(* Logix 5000 project; controller VET 1756-L62 rev 19.52; software revision 19.01; part 22 of 27 *)
(* tags used below, declared in another part *)
   _reset_local : ALIAS FOR _reset_locales.0;
   batch_in : batch;
   batch_out : batch;
   db1_var_batch : variables_procedimientos;
   db3_var_rep : variables_procedimientos;
   var_wd : variables_procedimientos;
   _Eqp_Cfg : Eqp_Cfg[800];
   Batch : batch[10];
   borrar : DINT[100];
   DRT : DRTs[10];
   simulacion : BOOL;
   TabBin : Bins_Setup;
   Timer : TIMER[500];
   vdf : VDFS[20];
(* Main, continued *)

ROUTINE main   (* ladder *)
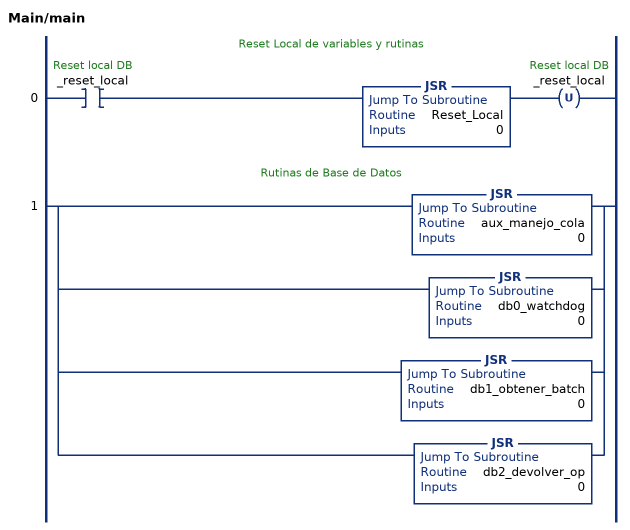
   // Reset Local de variables y rutinas
   0: XIC(_reset_local)JSR(Reset_Local,0)OTU(_reset_local);
   // Rutinas de Base de Datos
   1: [JSR(aux_manejo_cola,0) ,JSR(db0_watchdog,0) ,JSR(db1_obtener_batch,0) ,JSR(db2_devolver_op,0) ];
END_ROUTINE

ROUTINE Reset_Local   (* ladder *)
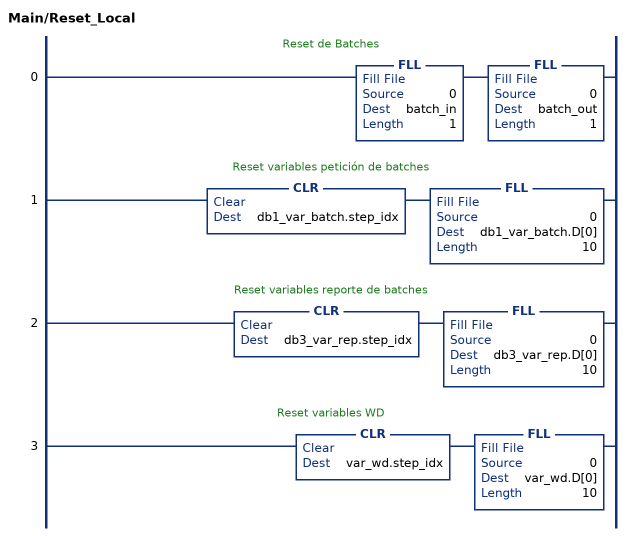
   // Reset de Batches
   0: FLL(0,batch_in,1)FLL(0,batch_out,1);
   // Reset variables petición de batches
   1: CLR(db1_var_batch.step_idx)FLL(0,db1_var_batch.D[0],10);
   // Reset variables reporte de batches
   2: CLR(db3_var_rep.step_idx)FLL(0,db3_var_rep.D[0],10);
   // Reset variables WD
   3: CLR(var_wd.step_idx)FLL(0,var_wd.D[0],10);
END_ROUTINE
END_PROGRAM

PROGRAM Main1   (* main routine Main, fault routine Error_Handler *)
VAR
   Automatismos : DINT := 7;
   Aux : DINT[500] := ([0] := 2014, [1] := 5, [2] := 15, [3] := 18, [4] := 46, [5] := 49, [6] := 20121005, [7] := 1184649, [8] := 1335329064, [9] := 2097152, [10] := 310798972, [11] := 326008, [13] := 1073741824, [14] := 4, [15] := 100, [16] := 180, [17] := 180, [18] := -25306, [19] := 1000000000, [20] := 1000000000, [21] := 1000000, [22] := 1099, [25] := 3, [27] := 164, [28] := 6347, [30] := 32, [34] := 111, [35] := 27, [36] := 10, [38] := 9, [45] := 4, [46] := 420, [47] := 14, [49] := 15999, [51] := 1, [52] := 10, [53] := 1, [54] := 1, [55] := 2, [56] := 47, [57] := 5, [58] := 6, [61] := 10, [62] := 1, [63] := 60, [64] := 1, [71] := 10, [72] := 1, [73] := 10, [74] := 1, [75] := 1, [81] := 2020, [88] := 99, [89] := 10, [90] := 2, [91] := 23450666, [93] := 1, [94] := 3, [98] := 1, [99] := 10,
        [100] := 10114, [101] := 1, [102] := 2, [107] := 2, [110] := 20, [112] := 10, [114] := 10, [115] := 10, [118] := 10, [131] := 70, [134] := 70, [146] := 2268, [147] := 22, [149] := 111, [150] := 105650, [151] := 1, [153] := 1, [154] := 1, [158] := 3, [165] := 1, [166] := 45, [167] := 1, [172] := -1, [173] := -1, [174] := -1, [175] := -1, [176] := -1, [177] := -1, [178] := 39, [182] := -1, [183] := -1, [184] := -1, [185] := -1, [186] := -1, [187] := -1, [189] := 28, [191] := 3, [200] := 5043, [201] := 3696, [202] := 4954, [203] := 3145, [204] := 69660, [205] := 1978, [206] := 233, [207] := 1977, [208] := 233, [209] := 1976, [210] := 233, [211] := 1976, [212] := 233, [213] := 1, [216] := 1, [219] := 1, [251] := 60, [253] := 4953, [255] := 5067, [257] := 20, [259] := 1280, [260] := 1408, [276] := 6,
        [277] := 1, [278] := 1, [279] := 18, [280] := 108, [281] := -1, [282] := -1, [283] := 2, [284] := 11, [285] := 110, [286] := 90, [287] := 96, [288] := 2, [289] := 11, [290] := 2048, [293] := 2048, [294] := 1451, [295] := 114, [298] := 114, [299] := 3543, [300] := 10, [301] := 1, [302] := 492, [303] := 493, [304] := 11, [314] := 7, [320] := 1, [321] := 16982, [322] := 10, [331] := 1, [333] := 10, [334] := 1980, [335] := 1, [345] := 10, [346] := 20, [347] := 3001, [351] := 7, [362] := 5, [365] := 10, [366] := 10, [367] := 3696, [370] := 10, [371] := 15, [372] := 20, [373] := 19, [380] := 18212712, [390] := 20, [391] := 299136, [392] := 11, [393] := 1, [394] := 1, [395] := 7, [399] := 757, [400] := 757, [401] := 757, [443] := 536870912, [450] := 1, [451] := 2, [452] := 4, [453] := 8, [454] := 16,
        [455] := 32, [456] := 64, [457] := 128, [458] := 256, [459] := 512, [460] := 1024, [461] := 2048, [462] := 4096, [463] := 8192, [464] := 16384, [465] := 32768, [466] := 65536, [467] := 131072, [468] := 262144, [469] := 524288, [470] := 1048576, [471] := 2097152, [472] := 4194304, [473] := 8388608, [474] := 16777216, [475] := 33554432, [476] := 67108864, [477] := 134217728, [478] := 268435456, [479] := 536870912, [480] := 1073741824, [481] := -2147483648);
        [345]   // Estado para Reporte. DMM en Bitácora
        [86]   // Estado para Import MP en Bitácora
        [137]   // Nº LiveBin vaciandose a Molienda
        [165]   // Estado para Error en Ingreso MP
        [270]   // Estado para Error en Ingreso MP
        [304]   // Estado para Escribir en Bitácora
        [164]   // Aux resumen timestamp rpt dmm
        [184]   // Auxiliar para username Mov MP
        [114]   // Status Control Nivel TOL-103-00
        [115]   // Status Control Nivel TOL-203-00
        [125]   // Status Start-Stop Mezcladora L1
        [258]   // Usuario Login Old Interfaz #10
        [50]   // Lugar de Dosif. de Prod sin Bin
        [121]   // Estado entre Tolva y livebins
        [190]   // Tipo Termino (1) Auto (2) Man
        [240]   // Usuario Login Old Interfaz #1
        [242]   // Usuario Login Old Interfaz #2
        [244]   // Usuario Login Old Interfaz #3
        [246]   // Usuario Login Old Interfaz #4
        [248]   // Usuario Login Old Interfaz #5
        [250]   // Usuario Login Old Interfaz #6
        [252]   // Usuario Login Old Interfaz #7
        [254]   // Usuario Login Old Interfaz #8
        [256]   // Usuario Login Old Interfaz #9
        [283]   // Tipo Termino (1) Auto (2) Man
        [314]   // Interfaz grabado en Bitacora
        [366]   // Cod Error Interno Batch Borrado
        [107]   // Linea elegida para descargar mixer
        [401]   // Numero Transacción from SQL OLD
        [411]   // Status Trigger SQL_Code -> Code
        [271]   // Estado para escribir buffer mov MP
        [288]   // Aux Tipo Termino (1) Auto (2) Man
        [333]   // Estado para Pet. Linea en Bitácora
        [9].19   // Mux32_19
        [9].20   // Mux32_20
        [9].21   // Mux32_21
        [9].22   // Mux32_22
        [150]   // Lugar de Dosif. de Prod sin Bin Micros
        [9].23   // Mux32_23
        [72].12   // _
        [72].16   // _
        [72].17   // _
        [72].18   // _
        [72].19   // _
        [365]   // Estado para Batch Borrado en Bitácora
        [72].20   // _
        [72].21   // _
        [9].24   // Mux32_24
        [72].22   // _
        [72].23   // _
        [72].24   // _
        [9].25   // Mux32_25
        [9].26   // Mux32_26
        [9].27   // Mux32_27
        [9].28   // Mux32_28
        [9].29   // Mux32_29
        [72].25   // _
        [72].26   // _
        [72].27   // _
        [105]   // Nivel para Mixer en Linea 1
        [72].28   // _
        [72].29   // _
        [73]   // Bin Grupo
        [106]   // Nivel para Mixer en Linea 2
        [74]   // Flag
        [75]   // Prioridad Bin
        [76]   // Codigo Producto.
        [77]   // Bin a Reemplazar
        [9].30   // Mux32_30
        [142]   // Indice Bin 1ra Prio Micros
        [148]   // Indice Bin 2da Prio Micros
        [182]   // Manejo Cola Reportes Mov MP
        [77].0   // _
        [77].1   // _
        [77].2   // _
        [77].4   // _
        [183]   // Manejo Cola Reportes Mov MP
        [9].31   // Mux32_31
        [89]   // Status para Termino Batch en Bitácora
        [280]   // Indice Destino Bin A Ruta 1
        [77].5   // _
        [80]   // Auxiliar en Setup
        [281]   // Indice Destino Bin B Ruta 1
        [282]   // Indice Destino Bin C Ruta 1
        [81]   // Auxiliar en Setup
        [285]   // Indice Destino Bin A Ruta 2
        [82]   // Report State
        [286]   // Indice Destino Bin B Ruta 2
        [83]   // Rpt Code
        [10]   // System Elapsed Time
        [84]   // Rpt Bin
        [329]   // Numero Transacción from SQL
        [85]   // Rpt Bin Group
        [93]   // Busqueda de Linea Batch
        [93].0   // Linea 1
        [93].1   // Linea 2
        [94]   // Last Line Rx
        [95]   // Status LiveBin #1
        [101]   // Nivel para LiveBin #1
        [399]   // Numero Transacción from SQL
        [102]   // Nivel para LiveBin #2
        [11]   // Total WeightTemp
        [103]   // Nivel para LiveBin #3
        [12]   // Old Formula Index
        [104]   // # LiveBin a Descargar
        [108]   // nivel envio batch l1
        [109]   // nivel envio batch l2
        [113].0   // Misma Guia
        [120]   // Estado Tolvas Macro
        [122]   // LiveBin Nº1 Status
        [12].0   // Reset Hsk
        [432]   // Status Transporte MAC -> LB
        [30]   // Status Lectura Corrientes VDF
        [99]   // Estado para Error en Batch Rx
        [127]   // Status Trasp. bajo Mixer #1
        [123]   // Status Molinos
        [12].1   // General Reset
        [12].2   // Sec_Hsk1
        [12].3   // Sec_Hsk2
        [188]   // Bits de cola reportes Mov MP
        [124]   // Descarga Micros
        [126]   // Status Mezcladora L1
        [392]   // Estado para Wdog en Bitacora
        [128]   // Estado Molienda
        [129]   // Estado Tolva TOL-031
        [130]   // Status Liquidos
        [131]   // Estado Molino #1
        [132]   // LiveBin Nº2 Status
        [133]   // LiveBin Nº3 Status
        [12].4   // Fast_Hsk
        [134]   // Estado Molino #2
        [136]   // Status TOL-056-00
        [13]   // Common Eqp Type
        [139]   // Status Eleccion Prebin
        [140]   // Estado Func. Mixer
        [14]   // Quantum Seg
        [141]   // Tot Bins x Prod Micros
        [15]   // Eqp x Ciclo
        [16]   // Mixer L1 espera
        [144]   // Flag Micros
        [17]   // Mixer L2 Espera
        [18].0   // _
        [145]   // Prioridad Bin
        [18].1   // _
        [146]   // Codigo Producto Micros
        [147]   // Bin a Reemplazar Micros
        [149]   // Prod Sin Bin Micro
        [151]   // Linea Dosificando Micros
        [152]   // Last Group End Micros
        [100]   // Estado para Conf. Batch Rx
        [153]   // Cycles Counter Micros
        [18].2   // _
        [18].3   // _
        [18].4   // _
        [18].5   // _
        [18].17   // _
        [18].18   // _
        [19].3   // _
        [20]   // 1LLLAAATTT
        [21]   // Numero Actual
        [22]   // Numero Total
        [23]   // L1 Level
        [24]   // L2 Level
        [26]   // Descarga Micros Status
        [31]   // Valor Num Dec.
        [33]   // Peticion Dosif Liq
        [34]   // Cod. a Reemp.
        [35]   // Bin a Reemp.
        [39]   // State CTolvas
        [40]   // Estado Dosif. Macros
        [41]   // Tot Bins x Prod
        [154]   // 7-LMG-1187 State
        [155]   // 8-ELV-498 State
        [156]   // Status Del Batch
        [160]   // Mix Batch State
        [166]   // Queue inlet Index
        [172]   // Corr. RED-705-00
        [173]   // Corr. RED-046-00
        [174]   // Corr. VEN-108-00
        [175]   // Corr. VEN-208-00
        [175].0   // Ora Lin #1 o 3
        [175].1   // Ora Lin #2 o 3
        [175].2   // Ora Lin #4
        [181]   // Index Report Out Mov MP
        [42]   // Indice Bin 1ra Prio
        [185]   // Auxiliar Interfaz Mov MP
        [187]   // Queue Report Count Mov MP
        [189]   // Index Report IN Mov MP
        [191]   // Last Line Rx
        [135]   // Status Start-Stop LiveBins
        [192]   // Item Guia
        [143]   // Bin Lugar de Dosif Micros
        [186]   // Queue report status Mov MP
        [305]   // Suma Cod_error en Bitacora
        [193]   // MP
        [312]   // User grabado en Bitacora
        [194]   // Bin
        [201]   // _
        [203]   // _
        [204].0   // _
        [204].1   // _
        [204].2   // _
        [0]   // Year
        [1]   // Month
        [2]   // Day
        [204].3   // _
        [204].4   // _
        [204].5   // _
        [204].6   // _
        [204].7   // _
        [204].10   // _
        [43]   // Bin Lugar de Dosif
        [3]   // Hour
        [44]   // Flag
        [204].11   // _
        [204].12   // _
        [4]   // Minute
        [204].13   // _
        [5]   // Second
        [45]   // Prioridad Bin
        [204].16   // _
        [204].17   // _
        [46]   // Codigo Producto.
        [205]   // _
        [208]   // _
        [209]   // _
        [210]   // _
        [6]   // Date(YYYYMMDD)
        [7]   // Time (1HHMMSS)
        [272]   // Bin
        [273]   // State Input MP
        [275]   // Usuario Aux
        [8]   // Current Time (Raw)
        [9]   // Mux32
        [9].0   // Mux32_0
        [9].1   // Mux32_1
        [9].2   // Mux32_2
        [276]   // Interfaz Aux
        [9].3   // Mux32_3
        [277]   // Aux Ruta(1o2)
        [278]   // Aux Limite Inferior
        [279]   // Aux Limite Superior
        [284]   // State Next Ruta 1
        [289]   // State Next Ruta 2
        [290]   // Timer hacia Bin A Ruta 1
        [291]   // Timer hacia Bin B Ruta 1
        [292]   // Timer hacia Bin C Ruta 1
        [293]   // Timer total Ruta 1
        [47]   // Bin a Reemplazar
        [295]   // Timer hacia Bin A Ruta 2
        [296]   // Timer hacia Bin B Ruta 2
        [9].4   // Mux32_4
        [297]   // Timer hacia Bin C Ruta 2
        [298]   // Timer total Ruta 2
        [299]   // Timer total Ruta 2
        [9].5   // Mux32_5
        [300]   // Queue report status
        [301]   // Queue Bitac Count
        [48]   // Indice Bin 2da Prio
        [9].7   // Mux32_7
        [9].8   // Mux32_8
        [9].9   // Mux32_9
        [49]   // Prod sin Bins
        [302]   // Index Bitac Out
        [303]   // Index Bitac. Inlet
        [316]   // Arg1 Bitácora
        [317]   // Arg2 Bitácora
        [318]   // Arg3 Bitácora
        [51]   // Linea Dosificando
        [52]   // Last Group End
        [53]   // Contador
        [54]   // Cycles Counter
        [60]   // L1 Batch State
        [61]   // Tot Bins x Prod
        [62]   // Indice Bin 1ra Prio
        [63]   // Bin Grupo
        [9].10   // Mux32_10
        [319]   // Arg4 Bitácora
        [323]   // Change Type from SQL
        [64]   // Flag
        [65]   // Prioridad Bin
        [65].16   // _
        [324]   // Change Arg 0 from SQL
        [325]   // Change Arg 1 from SQL
        [66]   // Codigo Producto.
        [326]   // Change Arg 2 from SQL
        [327]   // Change Arg 3 from SQL
        [328]   // Change Arg 4 from SQL
        [331]   // DBBatch Status
        [332]   // Cod Error Interno BatchRx
        [334]   // Last Folio Rx
        [335]   // Last Linea Rx
        [340]   // Batch Report State
        [341]   // Report Inlet Index
        [342]   // Queue Reports Count
        [67]   // Bin a Reemplazar
        [343]   // Index Report Out
        [67].0   // _
        [346]   // Cod Error Interno Reporte
        [347]   // Last Folio Tx
        [70]   // L1 Batch State
        [71]   // Tot Bins x Prod
        [72]   // Indice Bin 1ra Prio
        [72].0   // _
        [350]   // Status Login
        [351]   // Aux Idx Interfaz
        [360]   // Borrar Batch Status
        [361]   // Folio Batch Borrado
        [362]   // Index Batch Borrado
        [367]   // Last Folio Borrado
        [72].1   // _
        [72].2   // _
        [370]   // Mov MP Status
        [9].11   // Mux32_11
        [72].3   // _
        [72].4   // _
        [72].5   // _
        [72].6   // _
        [72].7   // _
        [72].8   // _
        [72].9   // _
        [72].10   // _
        [9].12   // Mux32_12
        [371]   // Mov MP Buffer Count
        [372]   // Mov Mp Index Out
        [373]   // Mov MP Index IN
        [390]   // Wdog State
        [9].13   // Mux32_13
        [391]   // Comm Error Counter
        [393]   // Change Type from SQL
        [394]   // Index Modificacion
        [400]   // Transaction to SQL
        [410]   // Status Updates
        [430]   // Status Tolva MACRO 1
        [431]   // Status Tolva MACRO 2
        [9].14   // Mux32_14
        [433]   // Status LB 2 Tolva056
        [9].15   // Mux32_15
        [9].16   // Mux32_16
        [9].17   // Mux32_17
        [9].18   // Mux32_18
        [72].11   // _
        [25]   // _
        [27]   // _
        [28]   // _
        [32]   // _
        [36]   // _
        [37]   // _
        [38]   // _
        [55]   // _
   aux_auto : BOOL;
   aux_tolva : DINT[2];
   EColor : DINT[1000] := ([1] := 1, [2] := 4, [3] := 65, [4] := 81, [5] := 1, [6] := 517, [7] := 19505, [8] := 19505, [10] := 593, [11] := 593, [12] := 593, [13] := 593, [14] := 593, [15] := 593, [20] := 4, [21] := 4, [22] := 4, [23] := 4, [24] := 4, [25] := 4, [26] := 4, [27] := 4, [28] := 4, [29] := 4, [30] := 4, [31] := 4, [32] := 4, [33] := 4, [34] := 4, [35] := 4, [40] := 81, [41] := 81, [42] := 81, [43] := 65, [44] := 65, [45] := 81, [46] := 65, [47] := 81, [48] := 81, [49] := 65, [50] := 81, [51] := 65, [52] := 81, [53] := 81, [54] := 81, [55] := 65, [60] := 4, [61] := 4, [62] := 4, [63] := 4, [64] := 4, [65] := 4, [66] := 4, [67] := 4, [68] := 4, [69] := 4, [70] := 4, [71] := 4, [72] := 4, [73] := 4,
        [74] := 4, [80] := 81, [81] := 65, [82] := 81, [83] := 65, [84] := 81, [85] := 65, [86] := 81, [87] := 81, [88] := 65, [89] := 81, [90] := 65, [91] := 81, [92] := 65, [93] := 81, [94] := 593, [100] := 593, [101] := 593, [102] := 593, [103] := 593, [104] := 593, [105] := 593, [110] := 4, [111] := 593, [112] := 4, [113] := 593, [114] := 4, [115] := 593, [116] := 4, [117] := 593, [118] := 593, [119] := 593, [120] := 4, [121] := 593, [123] := 65, [129] := 4, [130] := 29, [131] := 593, [132] := 4, [133] := 221, [134] := 221, [135] := 1, [136] := 1, [137] := 221, [138] := 1041, [140] := 4, [141] := 593, [150] := 4, [151] := 593, [152] := 4, [153] := 593, [154] := 593, [155] := 593, [156] := 593, [157] := 593, [158] := 593, [159] := 593, [160] := 593, [161] := 593, [162] := 593,
        [163] := 593, [164] := 593, [165] := 593, [166] := 593, [167] := 593, [168] := 593, [170] := 7, [171] := 2, [200] := 4, [201] := 529, [202] := 81, [205] := 4, [206] := 81, [207] := 81, [208] := 17, [209] := 4, [210] := 593, [211] := 81, [214] := 4, [215] := 81, [216] := 65, [217] := 4, [218] := 81, [219] := 65, [220] := 4, [221] := 81, [222] := 65, [223] := 4, [225] := 64, [226] := 529, [227] := 65, [228] := 65, [229] := 65, [230] := 65, [231] := 4, [232] := 529, [233] := 529, [234] := 4, [235] := 65, [236] := 4, [237] := 65, [239] := 529, [240] := 529, [241] := 529, [242] := 529, [243] := 529, [244] := 17, [245] := 17, [246] := 17, [247] := 4, [248] := 17, [251] := 65, [252] := 65, [253] := 529, [254] := 529, [255] := 536872196, [256] := 593, [257] := 65, [258] := 65, [259] := 537,
        [260] := 81, [261] := 67109381, [262] := 65, [263] := 65, [266] := 517, [268] := 528, [269] := 528, [270] := 67109377, [271] := 513, [272] := 513, [273] := 4, [290] := 4, [292] := 4, [294] := 4, [296] := 4, [301] := 4, [302] := 593, [303] := 593, [304] := 593, [305] := 4, [307] := 4, [308] := 65, [312] := 67109381, [314] := 65, [315] := 81, [316] := 12, [317] := 17, [318] := 529, [319] := 4, [320] := 65, [322] := 81, [323] := 529, [324] := 65, [325] := 81, [326] := 12, [327] := 17, [328] := 529, [329] := 132, [330] := 65, [332] := 81, [333] := 528, [334] := 65, [335] := 65, [336] := 81, [337] := 65, [338] := 65, [339] := 65, [340] := 1, [341] := 65, [342] := 529, [343] := 4, [344] := 593, [345] := 593, [346] := 593, [347] := 4, [349] := 260, [350] := 65, [354] := 1041, [356] := 65, [357] := 81,
        [358] := 12, [359] := 17, [360] := 529, [361] := 4, [362] := 65, [364] := 81, [365] := 536, [366] := 65, [367] := 81, [368] := 12, [369] := 17, [370] := 529, [371] := 4, [372] := 65, [374] := 81, [375] := 528, [376] := 65, [377] := 65, [378] := 81, [379] := 65, [380] := 65, [381] := 1089, [382] := 1, [383] := 1089, [384] := 529, [385] := 4, [386] := 65, [387] := 536871943, [388] := 529, [389] := 529, [390] := 529, [392] := 65, [393] := 529, [394] := 529, [395] := 536871943, [396] := 529, [398] := 81, [399] := 529, [400] := 529, [401] := 536871943, [402] := 536871943, [403] := 529, [404] := 529, [405] := 529, [406] := 529, [408] := 1, [409] := 529, [410] := 529, [411] := 529, [412] := 529, [413] := 529, [414] := 529, [415] := 529, [416] := 529, [418] := 81, [419] := 536871943, [420] := 536871943, [421] := 529, [422] := 529, [423] := 529,
        [424] := 529, [425] := 529, [426] := 529, [428] := 1, [429] := 529, [430] := 529, [431] := 529, [432] := 529, [433] := 529, [434] := 529, [435] := 529, [436] := 529, [438] := 4, [439] := 529, [440] := 4, [441] := 529, [442] := 260, [443] := 529, [444] := 4, [445] := 529, [446] := 4, [447] := 529, [448] := 4, [449] := 529, [450] := 260, [451] := 529, [452] := 260, [453] := 529, [454] := 260, [455] := 529, [456] := 4, [457] := 529, [458] := 4, [459] := 529, [460] := 4, [461] := 529, [462] := 4, [463] := 529, [464] := 4, [465] := 529, [466] := 4, [467] := 529, [468] := 4, [469] := 529, [601] := 17, [602] := 529, [603] := 529, [604] := 529, [605] := 529, [606] := 529, [607] := 529, [608] := 529, [609] := 1, [610] := 6, [611] := 81, [612] := 529, [613] := 529, [614] := 529, [615] := 529, [616] := 529,
        [617] := 529, [618] := 529, [619] := 1, [620] := 1, [621] := 4, [622] := 529, [623] := 4, [624] := 529, [625] := 4, [626] := 529, [701] := 4, [703] := 1, [704] := 1, [706] := 529, [707] := 529, [710] := 4, [711] := 4, [712] := 4, [720] := 1, [721] := 1, [827] := 2, [828] := 2, [829] := 1, [830] := 1);
   Eqp : Equipo[50] := ([0].S.Bits2 := 1146880, [1].Timer.Tpo1.PRE := 5000, [1].Timer.Tpo2.PRE := 5000, [1].Timer.Tpo3.PRE := 3000, [1].Timer.Tpo4.PRE := 10000, [1].Timer.Tpo4.EN := 1, [1].Timer.Tpo4.DN := 1, [1].Timer.Tpo5.PRE := 3000, [1].Timer.Tpo5.ACC := 3210, [1].Timer.Tpo5.EN := 1, [1].Timer.Tpo5.DN := 1, [1].Timer.Tpo6.PRE := 3000, [1].S.Bits1 := 81, [1].S.Bits2 := 2600960, [1].S.Bits3 := 1073807361, [1].Next := 171, [1].Color := 6, [2].Timer.Tpo1.PRE := 5000, [2].Timer.Tpo2.PRE := 5000, [2].Timer.Tpo3.PRE := 3000, [2].Timer.Tpo4.PRE := 10000, [2].Timer.Tpo5.PRE := 3000, [2].Timer.Tpo6.PRE := 3000, [2].S.Bits1 := 593, [2].S.Bits2 := 2600960, [2].S.Bits3 := 1073807361, [2].Next := 35, [2].Color := 2, [3].Timer.Tpo1.PRE := 5000, [3].Timer.Tpo2.PRE := 5000, [3].Timer.Tpo3.PRE := 3000, [3].Timer.Tpo4.PRE := 10000, [3].Timer.Tpo5.PRE := 3000, [3].Timer.Tpo6.PRE := 3000, [3].S.Bits1 := 1041, [3].S.Bits2 := 136810501, [4].Timer.Tpo1.PRE := 5000, [4].Timer.Tpo2.PRE := 5000, [4].Timer.Tpo3.PRE := 3000, [4].Timer.Tpo4.PRE := 10000, [4].Timer.Tpo5.PRE := 3000, [4].Timer.Tpo6.PRE := 3000, [4].S.Bits1 := 1024, [4].S.Bits2 := 368655, [5].Timer.Tpo1.PRE := 5000, [5].Timer.Tpo2.PRE := 5000, [5].Timer.Tpo3.PRE := 3000, [5].Timer.Tpo4.PRE := 10000, [5].Timer.Tpo5.PRE := 3000, [5].Timer.Tpo6.PRE := 3000, [5].S.Bits1 := 1077936290, [5].S.Bits2 := 335872, [5].S.Bits3 := 1073807361, [5].Next := 129, [5].Color := 5, [6].Timer.Tpo1.PRE := 5000, [6].Timer.Tpo2.PRE := 5000, [6].Timer.Tpo3.PRE := 3000, [6].Timer.Tpo4.PRE := 10000, [6].Timer.Tpo5.PRE := 3000,
        [6].Timer.Tpo6.PRE := 3000, [6].S.Bits1 := 593, [6].S.Bits2 := 2600960, [6].S.Bits3 := 1073807361, [6].Next := 35, [6].Color := 2, [7].Timer.Tpo1.PRE := 15000, [7].Timer.Tpo2.PRE := 15000, [7].Timer.Tpo3.PRE := 15000, [7].Timer.Tpo4.PRE := 20000, [7].Timer.Tpo4.EN := 1, [7].Timer.Tpo4.TT := 1, [7].Timer.Tpo5.PRE := 1000, [7].Timer.Tpo6.PRE := 1000, [7].S.Bits1 := 19505, [7].S.Bits2 := 2592768, [8].Timer.Tpo1.PRE := 5000, [8].Timer.Tpo2.PRE := 5000, [8].Timer.Tpo3.PRE := 3000, [8].Timer.Tpo4.PRE := 10000, [8].Timer.Tpo5.PRE := 3000, [8].Timer.Tpo6.PRE := 3000, [8].S.Bits1 := 4, [8].S.Bits2 := 1409024, [8].S.Bits3 := 16, [9].Timer.Tpo1.PRE := 5000, [9].Timer.Tpo2.PRE := 5000, [9].Timer.Tpo3.PRE := 3000, [9].Timer.Tpo4.PRE := 10000, [9].Timer.Tpo5.PRE := 3000, [9].Timer.Tpo6.PRE := 3000, [9].S.Bits2 := 1155072, [10].Timer.Tpo4.PRE := 10000, [10].Timer.Tpo5.PRE := 3000, [10].S.Bits1 := -32766, [10].S.Bits2 := 1277952, [10].Next := 77, [11].S.Bits2 := 1146880, [12].S.Bits2 := 1146880, [13].S.Bits2 := 1146880, [14].S.Bits2 := 1146880, [15].S.Bits2 := 1146880, [16].S.Bits2 := 1146880, [17].S.Bits2 := 1146880, [18].S.Bits2 := 1146880, [19].S.Bits2 := 1146880, [20].S.Bits2 := 1146880, [21].Timer.Tpo4.PRE := 10000, [21].Timer.Tpo4.EN := 1, [21].Timer.Tpo4.DN := 1, [21].Timer.Tpo5.PRE := 3000, [21].Timer.Tpo5.ACC := 3300, [21].Timer.Tpo5.EN := 1, [21].Timer.Tpo5.DN := 1, [21].S.Bits1 := 69, [21].S.Bits2 := 152272897, [21].S.Bits3 := 594192, [21].Next := 338, [21].Color := 2, [22].Timer.Tpo4.PRE := 10000,
        [22].Timer.Tpo4.EN := 1, [22].Timer.Tpo4.DN := 1, [22].Timer.Tpo5.PRE := 3000, [22].Timer.Tpo5.ACC := 3300, [22].Timer.Tpo5.EN := 1, [22].Timer.Tpo5.DN := 1, [22].S.Bits1 := 69, [22].S.Bits2 := 152272897, [22].S.Bits3 := 594192, [22].Next := 339, [22].Color := 2, [23].Timer.Tpo4.PRE := 10000, [23].Timer.Tpo4.EN := 1, [23].Timer.Tpo4.DN := 1, [23].Timer.Tpo5.PRE := 3000, [23].Timer.Tpo5.ACC := 3299, [23].Timer.Tpo5.EN := 1, [23].Timer.Tpo5.DN := 1, [23].S.Bits1 := 69, [23].S.Bits2 := 152272897, [23].S.Bits3 := 594192, [23].Next := 340, [23].Color := 2, [24].Timer.Tpo4.PRE := 10000, [24].Timer.Tpo4.EN := 1, [24].Timer.Tpo4.DN := 1, [24].Timer.Tpo5.PRE := 3000, [24].Timer.Tpo5.ACC := 3300, [24].Timer.Tpo5.EN := 1, [24].Timer.Tpo5.DN := 1, [24].S.Bits1 := 165, [24].S.Bits2 := 152272897, [24].S.Bits3 := 528400, [24].Next := 386, [24].Color := 5, [25].Timer.Tpo4.PRE := 10000, [25].Timer.Tpo4.EN := 1, [25].Timer.Tpo4.DN := 1, [25].Timer.Tpo5.PRE := 3000, [25].Timer.Tpo5.ACC := 3300, [25].Timer.Tpo5.EN := 1, [25].Timer.Tpo5.DN := 1, [25].S.Bits1 := 69, [25].S.Bits2 := 152272897, [25].S.Bits3 := 528400, [25].Next := 601, [25].Color := 2, [26].Timer.Tpo4.PRE := 10000, [26].Timer.Tpo4.TT := 1, [26].Timer.Tpo4.DN := 1, [26].Timer.Tpo5.PRE := 3000, [26].Timer.Tpo5.ACC := 3299, [26].Timer.Tpo5.EN := 1, [26].Timer.Tpo5.DN := 1, [26].S.Bits1 := 165, [26].S.Bits2 := 18063881, [26].S.Bits3 := 1074336051, [26].Next := 604, [26].Color := 5, [27].Timer.Tpo4.PRE := 10000,
        [27].Timer.Tpo4.EN := 1, [27].Timer.Tpo4.DN := 1, [27].Timer.Tpo5.PRE := 3000, [27].S.Bits1 := 65, [27].S.Bits2 := 152272896, [27].S.Bits3 := 594176, [27].Next := 338, [27].Color := 2, [28].Timer.Tpo4.PRE := 10000, [28].Timer.Tpo4.EN := 1, [28].Timer.Tpo4.DN := 1, [28].Timer.Tpo5.PRE := 3000, [28].S.Bits1 := 65, [28].S.Bits2 := 152272896, [28].S.Bits3 := 594176, [28].Next := 338, [28].Color := 2, [29].Timer.Tpo4.PRE := 10000, [29].Timer.Tpo4.EN := 1, [29].Timer.Tpo4.DN := 1, [29].Timer.Tpo5.PRE := 3000, [29].S.Bits1 := 65, [29].S.Bits2 := 152272896, [29].S.Bits3 := 594176, [29].Next := 338, [29].Color := 2, [30].Timer.Tpo1.PRE := 5000, [30].Timer.Tpo2.PRE := 5000, [30].Timer.Tpo3.PRE := 3000, [30].Timer.Tpo4.PRE := 10000, [30].Timer.Tpo5.PRE := 3000, [30].Timer.Tpo6.PRE := 3000, [30].S.Bits1 := 68, [30].S.Bits2 := 1146880, [30].S.Bits3 := 256, [30].Next := 150, [30].Color := 2, [31].Timer.Tpo4.PRE := 10000, [31].Timer.Tpo4.EN := 1, [31].Timer.Tpo4.DN := 1, [31].Timer.Tpo5.PRE := 3000, [31].S.Bits1 := 65, [31].S.Bits2 := 152272896, [31].S.Bits3 := 594176, [31].Next := 338, [31].Color := 2, [32].Timer.Tpo4.PRE := 10000, [32].Timer.Tpo4.EN := 1, [32].Timer.Tpo4.DN := 1, [32].Timer.Tpo5.PRE := 3000, [32].S.Bits1 := 65, [32].S.Bits2 := 152272896, [32].S.Bits3 := 594176, [32].Next := 338, [32].Color := 2, [33].Timer.Tpo4.PRE := 10000, [33].Timer.Tpo4.EN := 1, [33].Timer.Tpo4.DN := 1, [33].Timer.Tpo5.PRE := 3000, [33].S.Bits1 := 65,
        [33].S.Bits2 := 152272896, [33].S.Bits3 := 594176, [33].Next := 338, [33].Color := 2, [34].Timer.Tpo4.PRE := 10000, [34].Timer.Tpo4.EN := 1, [34].Timer.Tpo4.DN := 1, [34].Timer.Tpo5.PRE := 3000, [34].S.Bits1 := 65, [34].S.Bits2 := 152272896, [34].S.Bits3 := 594176, [34].Next := 338, [34].Color := 2, [35].Timer.Tpo4.PRE := 10000, [35].Timer.Tpo4.EN := 1, [35].Timer.Tpo4.DN := 1, [35].Timer.Tpo5.PRE := 3000, [35].S.Bits1 := 65, [35].S.Bits2 := 152272896, [35].S.Bits3 := 594176, [35].Next := 338, [35].Color := 2, [36].Timer.Tpo4.PRE := 10000, [36].Timer.Tpo4.EN := 1, [36].Timer.Tpo4.DN := 1, [36].Timer.Tpo5.PRE := 3000, [36].S.Bits1 := 65, [36].S.Bits2 := 152272896, [36].S.Bits3 := 594176, [36].Next := 338, [36].Color := 2, [37].Timer.Tpo4.PRE := 10000, [37].Timer.Tpo4.EN := 1, [37].Timer.Tpo4.DN := 1, [37].Timer.Tpo5.PRE := 3000, [37].S.Bits1 := 65, [37].S.Bits2 := 152272896, [37].S.Bits3 := 594176, [37].Next := 338, [37].Color := 2, [38].Timer.Tpo4.PRE := 10000, [38].Timer.Tpo4.EN := 1, [38].Timer.Tpo4.DN := 1, [38].Timer.Tpo5.PRE := 3000, [38].S.Bits1 := 65, [38].S.Bits2 := 152272896, [38].S.Bits3 := 594176, [38].Next := 338, [38].Color := 2, [39].Timer.Tpo4.PRE := 10000, [39].Timer.Tpo4.EN := 1, [39].Timer.Tpo4.DN := 1, [39].Timer.Tpo5.PRE := 3000, [39].S.Bits1 := 65, [39].S.Bits2 := 152272896, [39].S.Bits3 := 594177, [39].Next := 338, [39].Color := 2, [40].S.Bits2 := 1146880, [41].Timer.Tpo1.PRE := 5000,
        [41].Timer.Tpo2.PRE := 5000, [41].Timer.Tpo3.PRE := 3000, [41].Timer.Tpo4.PRE := 10000, [41].Timer.Tpo5.PRE := 3000, [41].Timer.Tpo6.PRE := 3000, [41].S.Bits1 := 593, [41].S.Bits2 := 1077385216, [41].S.Bits3 := 1073741825, [41].Color := 2, [42].S.Bits2 := 1146880, [43].S.Bits2 := 1146880, [44].S.Bits2 := 1146880, [45].S.Bits2 := 1146880, [46].S.Bits2 := 1146880, [47].S.Bits2 := 1146880, [48].S.Bits2 := 1146880, [49].S.Bits2 := 1146880);
        [2].STAT1.10   // _
        [2].STAT1.14   // _
        [2].STAT1.15   // _
        [2].STAT1.2   // _
        [2].STAT1.31   // _
        [2].STAT1.4   // _
        [2].STAT1.9   // _
        [2].STAT2.16   // _
        [2].STAT2.17   // _
        [2].STAT2.18   // _
        [2].STAT2.20   // _
        [2].STAT2.29   // _
        [2].STAT2.31   // _
        [2].STAT3.0   // _
        [2].STAT3.1   // _
        [2].STAT3.4   // _
        [2].STAT3.8   // _
        [3].BITS._1.0   // _
        [3].BITS._1.1   // _
        [3].BITS._1.10   // _
        [3].BITS._1.14   // _
        [3].BITS._1.15   // _
        [3].BITS._1.2   // _
        [3].BITS._1.4   // _
        [3].BITS._1.9   // _
        [3].BITS._2.16   // _
        [3].BITS._2.17   // _
        [3].BITS._2.18   // _
        [3].BITS._2.20   // _
        [3].BITS._2.21   // _
        [3].BITS._2.29   // _
        [3].BITS._2.31   // _
        [3].BITS._3.0   // _
        [3].BITS._3.1   // _
        [3].BITS._3.4   // _
        [3].BITS._3.5   // _
        [3].BITS._3.8   // _
        [3].BITS._3.9   // _
        [3].STAT1.0   // _
        [3].STAT1.1   // _
        [3].STAT1.10   // _
        [3].STAT1.14   // _
        [3].STAT1.15   // _
        [3].STAT1.2   // _
        [3].STAT1.4   // _
        [3].STAT1.9   // _
        [3].STAT2.16   // _
        [3].STAT2.17   // _
        [3].STAT2.18   // _
        [3].STAT2.20   // _
        [3].STAT2.21   // _
        [3].STAT2.29   // _
        [3].STAT2.31   // _
        [3].STAT3.0   // _
        [3].STAT3.1   // _
        [3].STAT3.4   // _
        [3].STAT3.5   // _
        [3].STAT3.8   // _
        [3].STAT3.9   // _
        [5].BITS._1.0   // _
        [5].BITS._1.1   // _
        [5].BITS._1.10   // _
        [5].BITS._1.14   // _
        [5].BITS._1.15   // _
        [5].BITS._1.2   // _
        [5].BITS._1.4   // _
        [5].BITS._1.9   // _
        [5].BITS._2.16   // _
        [5].BITS._2.17   // _
        [5].BITS._2.18   // _
        [5].BITS._2.20   // _
        [5].BITS._2.29   // _
        [5].BITS._2.31   // _
        [5].BITS._3.0   // _
        [5].BITS._3.1   // _
        [5].BITS._3.4   // _
        [5].BITS._3.8   // _
        [5].STAT1.0   // _
        [5].STAT1.1   // _
        [5].STAT1.10   // _
        [5].STAT1.14   // _
        [5].STAT1.15   // _
        [5].STAT1.2   // _
        [5].STAT1.4   // _
        [5].STAT1.9   // _
        [5].STAT2.16   // _
        [5].STAT2.17   // _
        [5].STAT2.18   // _
        [5].STAT2.20   // _
        [5].STAT2.29   // _
        [5].STAT2.31   // _
        [5].STAT3.0   // _
        [5].STAT3.1   // _
        [5].STAT3.4   // _
        [5].STAT3.8   // _
        [1].S.BITS2.21   // Enable Resumen
        [1].S.BITS2.23   // Test
        [1].S.BITS2.27   // Cmd Auto Run
        [1].S.BITS2.31   // Output Run
        [1].S.BITS3.14   // Suspend F2
        [2].S.BITS1.0   // Enable
        [2].S.BITS1.1   // Falla Resumen
        [2].S.BITS1.2   // Conf. Open
        [2].S.BITS1.4   // Conf. Close
        [2].S.BITS1.9   // Input Close
        [2].S.BITS1.10   // Input Open
        [2].S.BITS1.15   // Falla Open
        [2].S.BITS1.29   // Falla Close
        [2].S.BITS1.30   // Falla Open
        [2].S.BITS2.0   // Osr
        [4].S.BITS1.9   // Input Cen.
        [4].S.BITS1.10   // Input Der.
        [4].S.BITS1.28   // Falla Izq.
        [4].S.BITS1.29   // Falla Cen.
        [4].S.BITS1.30   // Falla Der.
        [4].S.BITS2.0   // Osr
        [4].S.BITS2.11   // Enc Izq.
        [4].S.BITS2.12   // Enc Cen.
        [2].S.BITS2.7   // Susp Code
        [4].S.BITS2.13   // Enc Der.
        [2].S.BITS2.8   // Susp_LH Ret
        [4].S.BITS2.14   // Suspended
        [4].S.BITS2.15   // Auto-Man Group
        [4].S.BITS2.16   // Enable Equipo
        [4].S.BITS2.17   // Enable Group
        [4].S.BITS2.18   // Enable Group
        [7].S.BITS1.10   // DRot Abajo
        [4].S.BITS2.20   // Reset Falla
        [4].S.BITS2.21   // Enable Resumen
        [4].S.BITS2.23   // Test
        [2].S.BITS2.12   // Enc Open
        [4].S.BITS2.25   // Cmd Auto Izq.
        [4].S.BITS2.26   // Cmd Auto Cen.
        [4].S.BITS2.27   // Cmd Auto Der.
        [4].S.BITS2.29   // Output Izq.
        [2].S.BITS2.13   // Enc Sgte
        [4].S.BITS2.30   // Output Cen.
        [4].S.BITS2.31   // Output Der.
        [2].S.BITS2.14   // Suspended
        [5].S.BITS1.0   // Enable
        [2].S.BITS2.15   // Auto-Man Group
        [2].S.BITS2.16   // Enable Equipo
        [5].S.BITS1.1   // Falla Resumen
        [5].S.BITS1.2   // Conf. Open
        [5].S.BITS1.4   // Conf. Close
        [5].S.BITS1.5   // Enable Resumen
        [5].S.BITS1.9   // Input Close
        [5].S.BITS1.10   // Input Open
        [5].S.BITS1.29   // Falla Close
        [5].S.BITS1.30   // Falla Open
        [5].S.BITS2.0   // Osr
        [5].S.BITS2.12   // Enc Open
        [5].S.BITS2.13   // Enc Sgte
        [2].S.BITS2.17   // Enable Group
        [5].S.BITS2.14   // Suspended
        [2].S.BITS2.18   // Enable Group
        [5].S.BITS2.15   // Auto-Man Group
        [5].S.BITS2.16   // Enable Equipo
        [5].S.BITS2.17   // Enable Group
        [5].S.BITS2.18   // Enable Group
        [2].S.BITS2.20   // Reset Falla
        [2].S.BITS2.21   // Enable Resumen
        [2].S.BITS2.23   // Test
        [5].S.BITS2.20   // Reset Falla
        [2].S.BITS2.27   // Cmd Auto Open
        [2].S.BITS2.29   // Osr
        [5].S.BITS2.23   // Test
        [5].S.BITS2.27   // Cmd Auto Open
        [5].S.BITS2.30   // Output Close
        [5].S.BITS2.31   // Output Open
        [2].S.BITS2.30   // Output Close
        [7].S.BITS1.0   // Enable
        [2].S.BITS2.31   // Output Open
        [3].S.BITS1.0   // Enable
        [1].S.BITS1.4   // Enable Resumen
        [3].S.BITS1.1   // Falla Resumen
        [3].S.BITS1.2   // Conf. Izq.
        [1].S.BITS1.7   // IVel 0
        [3].S.BITS1.4   // Conf. Der.
        [1].S.BITS1.8   // IAtoche
        [3].S.BITS1.9   // Input Izq.
        [1].S.BITS1.9   // IOverLoad
        [3].S.BITS1.10   // Input Der.
        [1].S.BITS1.10   // IConf. V0
        [1].S.BITS1.26   // Falla Bin Vacio
        [7].S.BITS1.1   // Falla Resumen
        [7].S.BITS1.2   // IConf Marcha
        [7].S.BITS1.3   // Conf. Mar. Auto
        [7].S.BITS1.4   // Enable Resumen
        [7].S.BITS1.9   // I Overload
        [7].S.BITS1.27   // Falla Movimiento
        [7].S.BITS1.28   // Falla Conf. Marcha
        [3].S.BITS1.29   // Falla Izq.
        [3].S.BITS1.30   // Falla Der.
        [7].S.BITS1.29   // Falla OL
        [7].S.BITS1.30   // Falla Marcha
        [7].S.BITS2.0   // Osr
        [1].S.BITS1.27   // Falla V0
        [7].S.BITS2.7   // Susp Code
        [7].S.BITS2.8   // Susp_LH Ret
        [7].S.BITS2.11   // Enc Ext1
        [7].S.BITS2.12   // Enc Prop
        [7].S.BITS2.13   // Enc Sgte
        [7].S.BITS2.14   // Suspended
        [3].S.BITS2.0   // Osr
        [7].S.BITS2.15   // Auto-Man Group
        [7].S.BITS2.16   // Enable Equipo
        [7].S.BITS2.17   // Enable Group
        [7].S.BITS2.18   // Enable System
        [7].S.BITS2.20   // Reset Falla
        [7].S.BITS2.21   // Enable Resumen
        [7].S.BITS2.23   // Test
        [7].S.BITS2.27   // Cmd Avanzar
        [1].S.BITS1.28   // Falla Atoche
        [7].S.BITS2.31   // Output Run
        [8].S.BITS1.2   // IConf. Marcha
        [8].S.BITS1.8   // ILL
        [8].S.BITS1.9   // ILM
        [8].S.BITS1.10   // I LH
        [8].S.BITS1.29   // Sound LH
        [8].S.BITS2.0   // OSR LH
        [1].S.BITS1.29   // Falla OL
        [1].S.BITS1.30   // Falla Marcha
        [40].S.BITS1.0   // Hab Eqp A
        [3].S.BITS2.11   // Enc Der.
        [40].S.BITS1.2   // Feedback Bin A
        [1].S.BITS2.0   // Osr
        [3].S.BITS2.12   // Enc Propio
        [1].S.BITS2.7   // Susp Code
        [1].S.BITS2.8   // Susp_LH Ret
        [40].S.BITS1.4   // Hab Eqp A
        [40].S.BITS1.11   // Falla Bin Vacio
        [41].S.BITS1.2   // Feedback Bin B
        [1].S.BITS2.10   // Enc Filtro
        [41].S.BITS1.4   // Hab Eqp B
        [41].S.BITS2.27   // Cmd Auto Run
        [1].BITS._1.0   // _
        [3].S.BITS2.13   // Enc Sgte
        [3].S.BITS2.14   // Suspended
        [3].S.BITS2.15   // Auto-Man Group
        [1].S.BITS2.11   // Enc Ext1
        [1].BITS._1.1   // _
        [1].S.BITS2.12   // Enc Prop
        [3].S.BITS2.16   // Enable Equipo
        [1].S.BITS2.13   // Enc Sgte
        [3].S.BITS2.17   // Enable Group
        [1].S.BITS2.14   // Suspended
        [1].BITS._1.10   // _
        [1].BITS._1.12   // _
        [1].BITS._1.13   // _
        [1].BITS._1.14   // _
        [1].BITS._1.15   // _
        [1].BITS._1.2   // _
        [1].BITS._1.3   // _
        [1].BITS._1.7   // _
        [1].BITS._1.8   // _
        [1].BITS._1.9   // _
        [1].BITS._2.16   // _
        [1].BITS._2.17   // _
        [1].BITS._2.18   // _
        [1].BITS._2.20   // _
        [1].BITS._2.29   // _
        [1].BITS._2.31   // _
        [1].BITS._3.0   // _
        [1].BITS._3.14   // _
        [1].BITS._3.4   // _
        [1].BITS._3.8   // _
        [1].STAT1.0   // _
        [1].STAT1.1   // _
        [1].STAT1.10   // _
        [1].STAT1.12   // _
        [1].STAT1.13   // _
        [1].STAT1.14   // _
        [7].S.BITS1.12   // Conf Abajo
        [1].STAT1.15   // _
        [1].STAT1.2   // _
        [1].STAT1.3   // _
        [1].STAT1.7   // _
        [1].S.BITS2.15   // Auto-Man Group
        [1].STAT1.8   // _
        [1].STAT1.9   // _
        [1].STAT2.16   // _
        [1].STAT2.17   // _
        [3].S.BITS2.18   // Enable Group
        [1].STAT2.18   // _
        [1].STAT2.20   // _
        [1].STAT2.29   // _
        [1].STAT2.31   // _
        [1].STAT3.0   // _
        [1].STAT3.14   // _
        [1].STAT3.4   // _
        [3].S.BITS2.20   // Reset Falla
        [3].S.BITS2.21   // Enable Resumen
        [1].STAT3.8   // _
        [2].BITS._1.0   // _
        [1].S.BITS2.16   // Enable Equipo
        [2].BITS._1.1   // _
        [2].BITS._1.10   // _
        [2].BITS._1.14   // _
        [3].S.BITS2.23   // Test
        [2].BITS._1.15   // _
        [2].BITS._1.2   // _
        [2].BITS._1.4   // _
        [2].BITS._1.9   // _
        [2].BITS._2.16   // _
        [2].BITS._2.17   // _
        [3].S.BITS2.25   // Cmd Auto Izq.
        [2].BITS._2.18   // _
        [2].BITS._2.20   // _
        [3].S.BITS2.26   // Cmd Auto Izq.
        [3].S.BITS2.27   // Cmd Auto Der.
        [1].S.BITS2.17   // Enable Group
        [2].BITS._2.29   // _
        [3].S.BITS2.29   // Output Izq.
        [2].BITS._2.31   // _
        [2].BITS._3.0   // _
        [3].S.BITS2.30   // Output Izq.
        [3].S.BITS2.31   // Output Der.
        [4].S.BITS1.0   // Enable
        [4].S.BITS1.1   // Falla Resumen
        [4].S.BITS1.2   // Conf. Izq.
        [1].S.BITS1.0   // Enable
        [1].S.BITS1.1   // Falla Resumen
        [2].BITS._3.1   // _
        [2].BITS._3.4   // _
        [2].BITS._3.8   // _
        [1].S.BITS2.18   // Enable System
        [1].S.BITS1.2   // IConf. Marcha
        [4].S.BITS1.3   // Conf. Cen.
        [2].STAT1.0   // _
        [1].S.BITS1.3   // Conf. Mar. Auto
        [2].STAT1.1   // _
        [4].S.BITS1.4   // Conf. Der.
        [4].S.BITS1.8   // Input Izq.
        [1].S.BITS2.20   // Reset Falla
        [7].S.BITS2.30   // Output Levantar
        [7].S.BITS1.13   // Conf Arriba
        [7].S.BITS1.11   // DRot Arriba
        [7].S.BITS2.26   // Comando Levantar
        [7].S.BITS2.22   // Test Levantar
   Errors : Fault_Register := (Time_Low := 1955766070, Time_High := 205779, Type := 4, Code := 20, Info[0] := 16#0000_0005, Info[1] := 16#0000_4a73, Info[2] := 16#0000_334d, Info[3] := 16#003a_5b18);
   I : Index := (a := 45, c := 299, g := 32, i := 27, j := 492, k := 6, l := 141, m := 5, n := 1, o := 1, p := 1, r := 8, s := 119, u := 2, v := 20, w := 18, x := 30, y := 200, z := 14, a1 := 50, b1 := 50, c1 := 50, d1 := 50, e1 := 50, f1 := 50, g1 := 4, i1 := 16, k1 := 1, l1 := 8, n1 := 5, o1 := 8, p1 := 164, q1 := 4, s1 := 1, t1 := 15, u1 := 50, v1 := 6, w1 := 7, x1 := 1, y1 := 19, z1 := 93, a2 := 15, b2 := 19, c2 := 15, d2 := 14, f2 := 19, g2 := 15, i2 := 14, k2 := 4, l2 := 11, n2 := 19, o2 := 11, p2 := 241, q2 := 10, r2 := 1, s2 := 8, t2 := 8, u2 := 1, v2 := 60, w2 := 61,
        x2 := 8, y2 := 2, z2 := 256, d3 := 14, f3 := 28, g3 := 14, i3 := 14, k3 := 5, n3 := 300, r3 := 31, s3 := 19);
        .G   // Correlativo en TabBin
        .A   // Eqp Fast Count
        .B   // Eqp Fast Index
        .C   // Eqp Norm Index
        .D   // Eqp Type
        .D.1   // Motor
        .D.2   // Gate
        .D.3   // Bifurcada
        .D.4   // Trifurc.
        .D.5   // Valvula
        .D.6   // Secciona Gate
        .D.7   // Dist.Rot.
        .D.8   // Tolva o Bin
        .E   // Eqp Type
        .F   // Eqp Type
        .H   // Selector Index
        .I   // Index Report Out
        .J   // Index Report Out Bitacora
        .K   // Index Report Out Report Batch
        .M   // Index Batch
        .N   // Origen Index
        .O   // PID Index
        .P   // PID Index
        .R   // Index BatCode
        .S   // Rpt. Inlet Index
        .T   // Idex Status Batch
        .U   // Index Batch
        .V   // Index Out MovMP
        .W   // Index Inlet MovMP
        .X   // Eqp Type
        .Z   // Index BIn
        .E1   // Ind. Ing. Liq
        .F1   // Bin Selected
        .G1   // SubIndice Prod #1
        .H1   // SubIndice Prod #2
        .I1   // SubIndice Prod #1
        .J1   // SubIndice Prod #2
        .K1   // Lugar/10
        .M1   // DRT: Indice Posiciones
        .N1   // Index Bin
        .O1   // Indice Ingrediente
        .Q1   // Index Bin A,B,C
        .R1   // Index Bin
        .S1   // Ruta 1 o 2
        .T1   // Index Eqp
        .U1   // Index Block Input
        .V1   // Index Eqp
        .W1   // Idx Next Eqp
        .X1   // Index Login
        .Z1   // Queue inlet Index
        .A2   // Indice Productos
        .B2   // Indice por Bin
        .C2   // Indice copia Prod.
        .D2   // SInd copia Prod #1
        .E2   // SInd copia Prod #2
        .G2   // SubIndice Prod #1
        .H2   // SubIndice Prod #2
        .I2   // SubIndice Prod #1
        .J2   // SubIndice Prod #2
        .O2   // Indice Ingrediente
        .Q2   // Index Bin sim
        .R2   // DRT: Indice ultima pos
        .S2   // DRT: Indice Posiciones
        .U2   // DRT: Nº Input Pos.
        .X2   // Ruta 1 o 2
        .Y2   // DRT: Indice de Eqp DRT's
        .N3   // Index Bin
        .O3   // Indice Ingrediente
   PID : PID_Struct := (Core.CTL := 67109760, Core.SWM := 1, Core.DVPA := 1, Core.PVLA := 1, Core.PVHA := 1, Core.SP := 220.0, Core.KP := 0.01, Core.KI := 1.e-04, Core.BIAS := 46.748608, Core.MAXS := 400.0, Core.MINS := 5.0, Core.SO := 50.0, Core.MAXO := 100.0, Core.UPD := 10.0, Core.ERR := 220.0, Core.OUT := 50.0, Core.MAXI := 400.0, Core.MINI := 5.0, Core.MAXCV := 100.0, Core.MAXTIE := 100.0, Core.DATA[0] := 2.6944313, Core.DATA[1] := 20.253164, Core.DATA[3] := 220.0, Core.DATA[4] := 220.0, Core.DATA[5] := 0.25316456, Core.DATA[6] := 1.0, Core.DATA[7] := 160.0, Core.DATA[8] := 0.01, Core.DATA[9] := 1.e-04, Core.DATA[11] := 0.01, Core.DATA[12] := 1.e-04, Core.DATA[15] := 1.0, Core.DATA[16] := 1.0, Status := 1879048202, Info.SP := 56, Info.CV := 50, SP := 220.0, CV := 50.0, Upd := 10.0, Kp := 0.01, Ki := 1.e-04, ENU_LL := 5.0, ENU_LH := 400.0, AO := 50);
        .STATUS.2   // PID Mode Auto (1) Man (0)
        .STATUS.0   // Auto Request Man (1) Auto (0)
        .CORE.SP   // Setpoint ENU
        .CORE.KP   // Proportional Gain
        .CORE.KI   // Integral Gain 1/Sec
        .CORE.KD   // Derivative Time Sec
        .CORE.MAXS   // ENU High Limit
        .CORE.MINS   // ENU Low Limit
        .CORE.DB   // Deadband ENU
        .CORE.SO   // Control Variable (0-100%)
        .CORE.UPD   // Loop Update Sec
        .STATUS.3   // PID Enabled
        .INFO.PV   // Process Variable 0-100%
        .INFO.SP   // Setpoint 0-100%
        .INFO.CV   // Control Variable (0-100%)
        .PV   // Process Variable ENU
        .CV   // Control Variable (0-100%)
        .STATUS.1   // Operator Request Man (1) Auto (0)
   RunHours : DINT[1000] := ([1] := 25114, [2] := 25505, [3] := 32, [4] := 25590, [5] := 25570, [7] := 1, [8] := 543, [20] := 32778, [22] := 44, [24] := 32043, [26] := 92, [28] := 506, [29] := 13973, [30] := 33203, [31] := 33533, [32] := 21730, [33] := 9, [34] := 2, [40] := 14011, [41] := 14273, [42] := 26, [43] := 29296, [44] := 205, [45] := 32282, [46] := 15590, [47] := 22103, [48] := 23327, [49] := 441, [50] := 233, [52] := 1, [53] := 22814, [54] := 28, [55] := 6996, [60] := 74, [61] := 23538, [62] := 23541, [63] := 23555, [64] := 14248, [65] := 278, [66] := 254, [67] := 23734, [68] := 23751, [69] := 23769, [70] := 12366, [71] := 184, [72] := 230, [73] := 23040, [80] := 25116, [81] := 6, [82] := 30, [83] := 201, [84] := 176, [87] := 1, [88] := 2, [89] := 14, [90] := 3, [91] := 27, [92] := 48, [93] := 73, [101] := 56,
        [102] := 1500, [103] := 108, [104] := 626, [105] := 170, [110] := 524, [111] := 10, [112] := 786, [113] := 17, [114] := 2312, [115] := 20, [116] := 482, [117] := 3, [118] := 241, [119] := 36, [120] := 1090, [121] := 5, [123] := 8, [130] := 3326, [133] := 1201, [134] := 159, [135] := 108, [136] := 1117, [137] := 1087, [138] := 10, [140] := 396, [141] := 10390, [150] := 8049, [151] := 8, [170] := 3, [171] := 24689, [200] := 371, [201] := 177, [202] := 2170, [206] := 2334, [207] := 24862, [208] := 24208, [209] := 1235, [210] := 148, [211] := 24843, [214] := 6, [215] := 843, [216] := 647, [217] := 129, [218] := 307, [219] := 143, [220] := 139, [221] := 2685, [222] := 1344, [223] := 1412, [225] := 25645, [226] := 107, [227] := 24119, [228] := 24877, [229] := 24901, [230] := 24985, [231] := 19, [232] := 3, [233] := 20, [235] := 24986, [236] := 846,
        [237] := 25041, [239] := 925, [240] := 1228, [241] := 1203, [243] := 16, [244] := 2180, [245] := 1940, [246] := 1889, [247] := 1199, [248] := 703, [251] := 414, [252] := 489, [253] := 19, [254] := 154, [255] := 69, [256] := 12, [257] := 257, [258] := 275, [260] := 263, [261] := 19, [262] := 615, [263] := 389, [266] := 65, [267] := 295, [271] := 1087, [272] := 242, [290] := 36, [302] := 664, [303] := 212, [305] := 586, [307] := 5, [308] := 9891, [312] := 4, [314] := 24297, [315] := 24192, [316] := 451, [317] := 8463, [319] := 73, [320] := 24351, [322] := 24384, [323] := 418, [324] := 23747, [325] := 23749, [326] := 496, [327] := 11821, [328] := 491, [329] := 656, [330] := 23930, [332] := 23779, [333] := 2, [334] := 24779, [335] := 24792, [336] := 24701, [337] := 24241, [338] := 24379, [339] := 24588, [340] := 23534, [341] := 23867, [342] := 483, [343] := 556,
        [344] := 826, [345] := 135, [346] := 5, [347] := 761, [349] := 28, [350] := 10223, [356] := 23913, [357] := 23795, [358] := 810, [359] := 9681, [360] := 729, [361] := 238, [362] := 23615, [364] := 23691, [365] := 6, [366] := 23403, [367] := 23414, [368] := 4, [369] := 7555, [370] := 107, [371] := 95, [372] := 23352, [374] := 23625, [375] := 219, [376] := 24080, [377] := 24088, [378] := 24450, [379] := 23947, [380] := 23709, [381] := 23926, [382] := 23044, [383] := 23186, [384] := 476, [385] := 266, [386] := 24629, [387] := 210, [388] := 258, [389] := 448, [390] := 126, [392] := 23965, [393] := 59, [394] := 2, [396] := 124, [398] := 12500, [399] := 5, [400] := 249, [401] := 257, [402] := 250, [403] := 321, [404] := 245, [406] := 78, [408] := 12504, [412] := 82, [414] := 246, [415] := 79, [418] := 11241, [424] := 222, [428] := 12052, [434] := 170, [438] := 315,
        [443] := 20, [452] := 1, [460] := 47, [467] := 21, [704] := 4, [720] := 2, [721] := 2);
   RunSegs : DINT[1000] := ([1] := 2315, [2] := 2505, [3] := 2710, [4] := 2440, [5] := 2975, [6] := 2515, [7] := 1795, [8] := 2565, [20] := 1780, [22] := 400, [23] := 3040, [24] := 1920, [26] := 15, [28] := 2250, [29] := 3430, [30] := 1345, [31] := 545, [32] := 960, [33] := 235, [34] := 3175, [35] := 810, [40] := 2995, [41] := 920, [42] := 3290, [43] := 2865, [44] := 995, [45] := 2965, [46] := 2280, [47] := 2255, [48] := 3555, [49] := 3505, [50] := 2410, [51] := 2600, [52] := 3515, [53] := 1405, [54] := 1025, [55] := 800, [60] := 2475, [61] := 1640, [62] := 480, [63] := 805, [64] := 1145, [65] := 1960, [66] := 985, [67] := 3395, [68] := 3385, [69] := 2165, [70] := 1900, [71] := 1405, [72] := 2760, [73] := 815, [80] := 1765, [81] := 405, [82] := 2520, [83] := 2555, [84] := 2450, [85] := 2310, [86] := 345, [87] := 635, [88] := 45,
        [89] := 2950, [90] := 775, [91] := 465, [92] := 2445, [93] := 480, [101] := 2125, [102] := 2545, [103] := 1310, [104] := 2340, [105] := 3095, [110] := 2340, [111] := 2485, [112] := 2190, [113] := 3320, [114] := 3520, [115] := 1650, [116] := 2140, [117] := 480, [118] := 1505, [119] := 3580, [120] := 3545, [121] := 2640, [123] := 3080, [130] := 2135, [133] := 1200, [134] := 130, [135] := 2875, [136] := 2160, [137] := 235, [138] := 1225, [140] := 1490, [141] := 3370, [150] := 1780, [151] := 1645, [170] := 1290, [171] := 3365, [200] := 2820, [201] := 140, [202] := 1665, [206] := 2810, [207] := 2395, [208] := 25, [209] := 615, [210] := 1820, [211] := 650, [214] := 2355, [215] := 1510, [216] := 2525, [217] := 105, [218] := 120, [219] := 1975, [220] := 170, [221] := 1690, [222] := 850, [223] := 1050, [225] := 2895, [226] := 2990, [227] := 2335, [228] := 1210, [229] := 3240,
        [230] := 1615, [231] := 2250, [232] := 75, [233] := 1135, [234] := 3530, [235] := 1020, [236] := 1500, [237] := 335, [239] := 560, [240] := 1865, [241] := 2965, [242] := 510, [243] := 2165, [244] := 3210, [245] := 1315, [246] := 290, [247] := 2340, [248] := 3545, [251] := 3400, [252] := 755, [253] := 3055, [254] := 395, [255] := 2375, [256] := 2810, [257] := 760, [258] := 2655, [259] := 465, [260] := 160, [261] := 2735, [262] := 935, [263] := 2305, [266] := 745, [267] := 1355, [270] := 2260, [271] := 2470, [272] := 495, [290] := 1655, [292] := 2570, [294] := 3490, [301] := 5, [302] := 680, [303] := 2680, [304] := 2425, [305] := 2125, [307] := 1770, [308] := 2305, [312] := 600, [314] := 15, [315] := 510, [316] := 3105, [317] := 1775, [319] := 1730, [320] := 2545, [322] := 2855, [323] := 3155, [324] := 2755, [325] := 1700, [326] := 3230, [327] := 755, [328] := 210,
        [329] := 2795, [330] := 1795, [332] := 1190, [333] := 975, [334] := 945, [335] := 1565, [336] := 3330, [337] := 1350, [338] := 1570, [339] := 280, [340] := 1345, [341] := 2910, [342] := 405, [343] := 1450, [344] := 3165, [345] := 355, [346] := 655, [347] := 740, [349] := 2865, [350] := 235, [354] := 15, [356] := 1900, [357] := 2315, [358] := 3000, [359] := 1080, [360] := 1450, [361] := 3095, [362] := 120, [364] := 1650, [365] := 3465, [366] := 2370, [367] := 550, [368] := 735, [369] := 1455, [370] := 2860, [371] := 2785, [372] := 2175, [374] := 45, [375] := 1865, [376] := 2885, [377] := 2820, [378] := 45, [379] := 845, [380] := 1415, [381] := 2895, [382] := 1810, [383] := 1975, [384] := 130, [385] := 3340, [386] := 580, [387] := 815, [388] := 1195, [389] := 1555, [390] := 3290, [392] := 2770, [393] := 700, [394] := 855, [396] := 2010, [398] := 690, [399] := 1475,
        [400] := 1845, [401] := 2660, [402] := 1785, [403] := 930, [404] := 830, [406] := 1475, [408] := 495, [409] := 60, [410] := 250, [412] := 2805, [414] := 680, [415] := 2480, [416] := 60, [418] := 1510, [419] := 2005, [421] := 1125, [424] := 2890, [428] := 1130, [433] := 185, [434] := 850, [436] := 20, [438] := 1900, [441] := 5, [442] := 30, [443] := 1200, [444] := 35, [447] := 45, [450] := 820, [451] := 1200, [452] := 590, [460] := 3525, [461] := 10, [462] := 50, [464] := 1785, [467] := 800, [601] := 20, [611] := 10, [703] := 300, [704] := 2475, [720] := 1020, [721] := 980);
   RunStarts : DINT[1000] := ([1] := 6050, [2] := 2058, [3] := 557, [4] := 2470, [5] := 2399, [6] := 1256, [7] := 906, [8] := 356, [10] := 1, [11] := 6, [12] := 1, [13] := 2, [14] := 1, [15] := 1, [20] := 5674, [21] := 296, [22] := 181, [23] := 669, [24] := 5603, [25] := 1743, [26] := 666, [27] := 183, [28] := 75, [29] := 38308, [30] := 7803, [31] := 6208, [32] := 6670, [33] := 3808, [34] := 273, [35] := 614, [40] := 9552, [41] := 3715, [42] := 484, [43] := 4066, [44] := 348, [45] := 8669, [46] := 9009, [47] := 8827, [48] := 9180, [49] := 3032, [50] := 6311, [51] := 2435, [52] := 5151, [53] := 7532, [54] := 1018, [55] := 5621, [60] := 2233, [61] := 1790, [62] := 1580, [63] := 1658, [64] := 10612, [65] := 149, [66] := 3354, [67] := 1844, [68] := 1654, [69] := 1660, [70] := 11048, [71] := 1274, [72] := 905, [73] := 2715,
        [80] := 3218, [81] := 15070, [82] := 13076, [83] := 5589, [84] := 207, [85] := 6, [86] := 92, [87] := 40, [88] := 121, [89] := 1668, [90] := 124, [91] := 1630, [92] := 85, [93] := 3746, [94] := 21, [100] := 56, [101] := 8800, [102] := 101022, [103] := 3374, [104] := 31174, [105] := 3753, [110] := 23706, [111] := 989, [112] := 59173, [113] := 492, [114] := 125270, [115] := 543, [116] := 69995, [117] := 282, [118] := 17912, [119] := 1014, [120] := 154778, [121] := 337, [123] := 236, [130] := 153081, [131] := 64, [133] := 1058, [134] := 418, [135] := 127646, [136] := 126537, [137] := 128938, [138] := 129999, [140] := 1512, [141] := 31301, [150] := 25869, [151] := 2790, [153] := 66, [154] := 16, [155] := 46, [156] := 6, [157] := 22, [158] := 44, [159] := 3, [160] := 38, [161] := 66, [162] := 2, [163] := 44, [164] := 2, [165] := 22, [166] := 52,
        [167] := 2, [168] := 40, [170] := 162, [171] := 5492, [200] := 132, [201] := 124961, [202] := 125835, [206] := 153, [207] := 2533, [208] := 19448, [209] := 391, [210] := 128414, [211] := 5218, [214] := 1942, [215] := 42324, [216] := 44980, [217] := 75, [218] := 15176, [219] := 11496, [220] := 233, [221] := 64920, [222] := 59215, [223] := 8256, [225] := 3619, [226] := 126194, [227] := 67365, [228] := 5362, [229] := 3933, [230] := 2508, [231] := 2872, [232] := 2127, [233] := 4144, [234] := 2458, [235] := 3804, [236] := 1795, [237] := 5523, [239] := 36692, [240] := 29205, [241] := 33024, [242] := 28874, [243] := 3490, [244] := 12145, [245] := 1497, [246] := 4734, [247] := 1992, [248] := 4715, [251] := 3193, [252] := 986, [253] := 5257, [254] := 651, [255] := 3685, [256] := 3357, [257] := 7328, [258] := 3233, [259] := 382, [260] := 3314, [261] := 1118, [262] := 859, [263] := 4523, [266] := 2431,
        [267] := 2737, [268] := 79321, [269] := 10, [270] := 2506, [271] := 728, [272] := 4331, [290] := 27, [292] := 37, [294] := 187, [296] := 10, [299] := 205, [301] := 15, [302] := 462965, [303] := 461068, [304] := 462981, [305] := 261, [307] := 63, [308] := 70425, [312] := 96045, [314] := 1341, [315] := 1288, [316] := 117, [317] := 467304, [318] := 9454, [319] := 18, [320] := 1372, [322] := 11018, [323] := 60072, [324] := 11526, [325] := 1852, [326] := 825, [327] := 312126, [328] := 54090, [329] := 168, [330] := 2046, [332] := 2002, [333] := 64048, [334] := 1381, [335] := 1021, [336] := 1306, [337] := 11660, [338] := 9940, [339] := 4869, [340] := 8782, [341] := 1358, [342] := 303, [343] := 43159, [344] := 395666, [345] := 396120, [346] := 396575, [347] := 221, [349] := 12, [350] := 106290, [354] := 9838, [356] := 2104, [357] := 2055, [358] := 43414, [359] := 213018, [360] := 8369, [361] := 264,
        [362] := 1655, [364] := 1276, [365] := 47997, [366] := 14218, [367] := 14295, [368] := 162, [369] := 301753, [370] := 7730, [371] := 654, [372] := 1628, [374] := 1455, [375] := 52489, [376] := 975, [377] := 1193, [378] := 1130, [379] := 8441, [380] := 8056, [381] := 4185, [382] := 4123, [383] := 13206, [384] := 421, [385] := 102, [386] := 5203, [387] := 1299, [388] := 3512, [389] := 1298, [390] := 1515, [392] := 4196, [393] := 8166, [394] := 1050, [395] := 1027, [396] := 1102, [398] := 3796, [399] := 963, [400] := 1710, [401] := 667, [402] := 604, [403] := 736, [404] := 706, [405] := 745, [406] := 920, [408] := 3802, [409] := 781, [410] := 806, [411] := 761, [412] := 750, [413] := 640, [414] := 790, [415] := 742, [416] := 856, [418] := 3525, [419] := 691, [420] := 640, [421] := 687, [422] := 731, [423] := 570, [424] := 726, [425] := 644, [426] := 850, [428] := 3847,
        [429] := 740, [430] := 723, [431] := 716, [432] := 719, [433] := 704, [434] := 908, [435] := 739, [436] := 897, [438] := 150, [439] := 39, [440] := 111, [441] := 60, [442] := 85, [443] := 61, [444] := 251, [445] := 49, [446] := 101, [447] := 405, [448] := 108, [449] := 414, [450] := 102, [451] := 6, [452] := 13, [453] := 281, [454] := 2, [455] := 7, [456] := 9, [457] := 4, [458] := 8, [459] := 18, [460] := 14, [461] := 10, [462] := 10, [463] := 7, [464] := 21, [465] := 16, [466] := 6, [467] := 18, [468] := 19, [469] := 7, [601] := 1, [602] := 3, [603] := 5, [604] := 6, [605] := 3, [606] := 3, [607] := 3, [608] := 4, [611] := 1, [612] := 3, [613] := 3, [614] := 4, [615] := 5, [616] := 3, [617] := 3, [618] := 3, [623] := 1, [703] := 6, [704] := 4, [720] := 10,
        [721] := 15);
   String : STRING[40] := ([0] := '20140515', [1] := '1184649', [2] := '120140515184649', [3] := '                   _', [4] := '0', [5] := '1000010000011099', [6] := '1000000000                   _', [7] := '1                   _000000000                   _', [8] := '1                    _                  _000000000                   _', [9] := '1  0                  _                  _000000000                   _', [10] := '20140515184649', [11] := '0                  _               ', [12] := '0                  _               0', [13] := '0', [14] := '05020105354043313560200523092002157050059', [15] := '1002', [16] := '16', [17] := '10', [20] := '                   _', [21] := '10030050207CLC                   _', [22] := '0030050207CLC    ', [23] := '1000000000', [24] := ' $00$00$00 $00$00$00 $00$00$00 $00$00$00 $00$00$00 $00$00$00 $00$00$00 $00$00$00', [25] := '111002016099ECL1021', [26] := 'TOL ', [27] := 'ABRT', [28] := ' $00$00$00 $00$00$00 $00$00$00 $00$00$00 $00$00$00 $00$00$00 $00$00$00 $00$00$00', [29] := ' ', [30] := 'OK  ', [31] := 'INGR', [32] := 'ABRT', [33] := 'TOLV', [34] := 'NEQ ', [35] := 'RCTA', [36] := 'LOAD', [37] := ' $00$00$00 $00$00$00 $00$00$00 $00$00$00 $00$00$00 $00$00$00 $00$00$00 $00$00$00', [38] := '        ', [39] := '                   _');
        [8].LEN   // _
        [20]   // 1LLLAAATTT FFFFFFF
        [21]   // LLLAAATTT FFFFFFF
        [22]   // LLLAAATTT FFFFFFFSSSS
        [7]   // _
        [9]   // _
        [11]   // _
        [12]   // _
        [13]   // _
        [14]   // _
        [15]   // _
        [16]   // _
        [17]   // _
        [18]   // _
        [19]   // _
   TabEqp : INT[500] := ([0] := 7, [1] := 8, [2] := 40, [3] := 41, [4] := 42, [5] := 43, [6] := 44, [7] := 45, [8] := 46, [9] := 47, [10] := 48, [11] := 49, [12] := 50, [13] := 51, [14] := 52, [15] := 53, [16] := 54, [17] := 55, [18] := 80, [19] := 81, [20] := 82, [21] := 83, [22] := 84, [23] := 85, [24] := 86, [25] := 87, [26] := 88, [27] := 89, [28] := 90, [29] := 91, [30] := 92, [31] := 93, [32] := 94, [33] := 100, [34] := 101, [35] := 102, [36] := 103, [37] := 104, [38] := 105, [39] := 111, [40] := 113, [41] := 115, [42] := 117, [43] := 118, [44] := 119);
END_VAR

ROUTINE _Cntrl_Bifurc   (* ladder *)
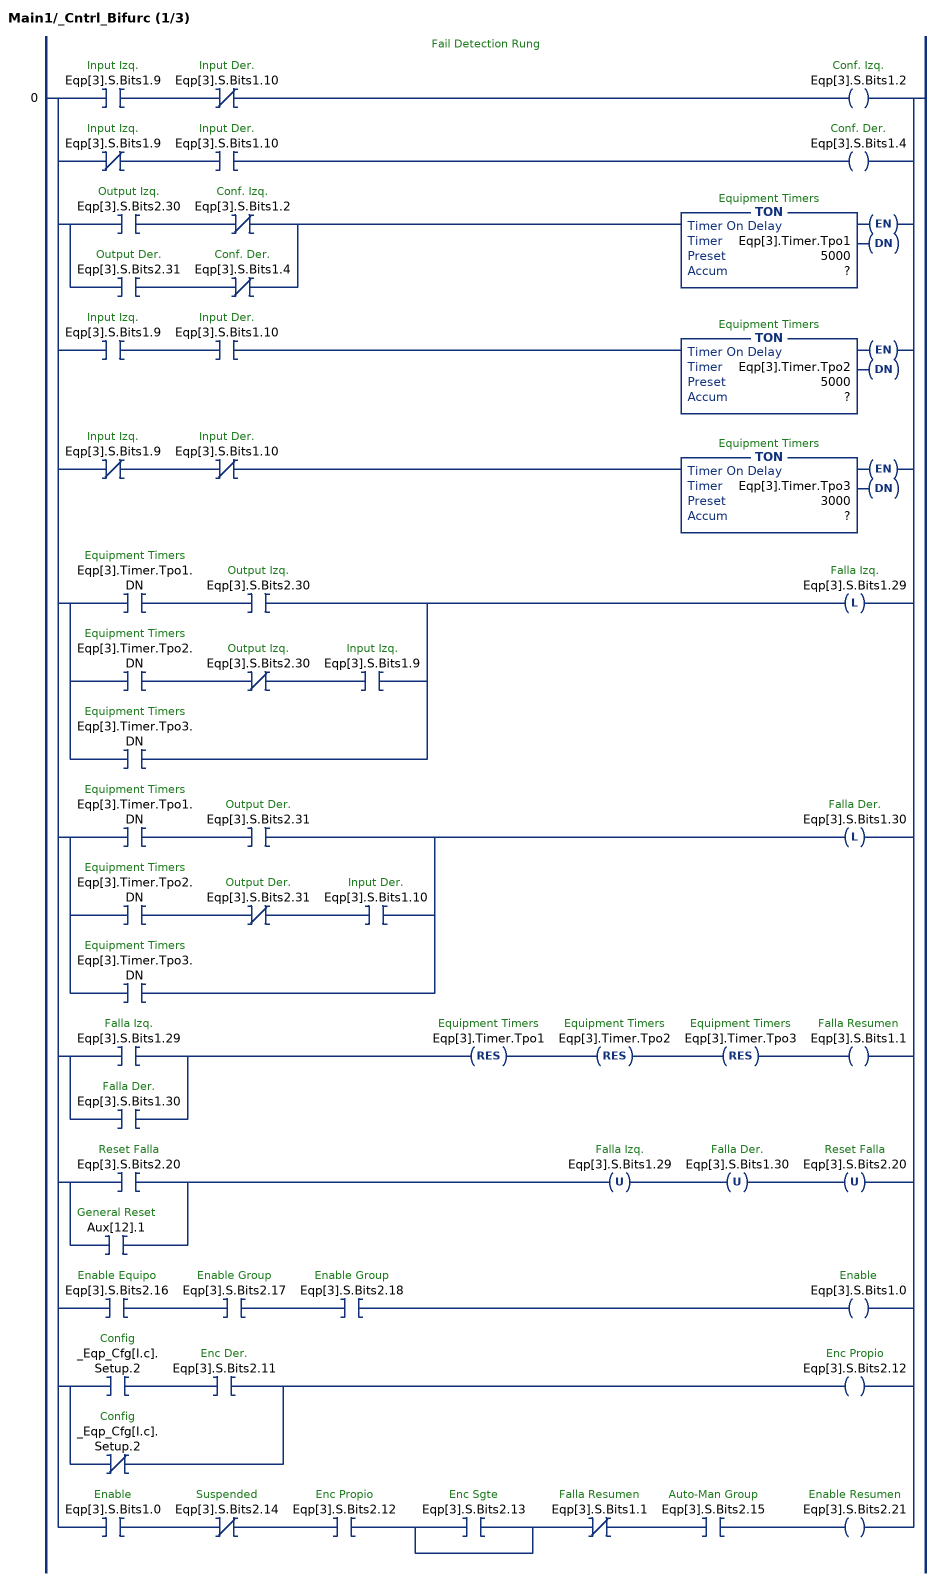
   // Fail Detection Rung
   0: [[XIC(Eqp[3].S.Bits1.9) XIO(Eqp[3].S.Bits1.10) OTE(Eqp[3].S.Bits1.2) ,XIO(Eqp[3].S.Bits1.9) XIC(Eqp[3].S.Bits1.10) OTE(Eqp[3].S.Bits1.4) ] ,[XIC(Eqp[3].S.Bits2.30) XIO(Eqp[3].S.Bits1.2) ,XIC(Eqp[3].S.Bits2.31) XIO(Eqp[3].S.Bits1.4) ] TON(Eqp[3].Timer.Tpo1,?,?) ,XIC(Eqp[3].S.Bits1.9) XIC(Eqp[3].S.Bits1.10) TON(Eqp[3].Timer.Tpo2,?,?) ,XIO(Eqp[3].S.Bits1.9) XIO(Eqp[3].S.Bits1.10) TON(Eqp[3].Timer.Tpo3,?,?) ,[XIC(Eqp[3].Timer.Tpo1.DN) XIC(Eqp[3].S.Bits2.30) ,XIC(Eqp[3].Timer.Tpo2.DN) XIO(Eqp[3].S.Bits2.30) XIC(Eqp[3].S.Bits1.9) ,XIC(Eqp[3].Timer.Tpo3.DN) ] OTL(Eqp[3].S.Bits1.29) ,[XIC(Eqp[3].Timer.Tpo1.DN) XIC(Eqp[3].S.Bits2.31) ,XIC(Eqp[3].Timer.Tpo2.DN) XIO(Eqp[3].S.Bits2.31) XIC(Eqp[3].S.Bits1.10) ,XIC(Eqp[3].Timer.Tpo3.DN) ] OTL(Eqp[3].S.Bits1.30) ,[XIC(Eqp[3].S.Bits1.29) ,XIC(Eqp[3].S.Bits1.30) ] RES(Eqp[3].Timer.Tpo1) RES(Eqp[3].Timer.Tpo2) RES(Eqp[3].Timer.Tpo3) OTE(Eqp[3].S.Bits1.1) ,[XIC(Eqp[3].S.Bits2.20) ,XIC(Aux[12].1) ] OTU(Eqp[3].S.Bits1.29) OTU(Eqp[3].S.Bits1.30) OTU(Eqp[3].S.Bits2.20) ,XIC(Eqp[3].S.Bits2.16) XIC(Eqp[3].S.Bits2.17) XIC(Eqp[3].S.Bits2.18) OTE(Eqp[3].S.Bits1.0) ,[XIC(_Eqp_Cfg[I.c].Setup.2) XIC(Eqp[3].S.Bits2.11) ,XIO(_Eqp_Cfg[I.c].Setup.2) ] OTE(Eqp[3].S.Bits2.12) ,XIC(Eqp[3].S.Bits1.0) XIO(Eqp[3].S.Bits2.14) XIC(Eqp[3].S.Bits2.12) [XIC(Eqp[3].S.Bits2.13) ,] XIO(Eqp[3].S.Bits1.1) XIC(Eqp[3].S.Bits2.15) OTE(Eqp[3].S.Bits2.21) ];
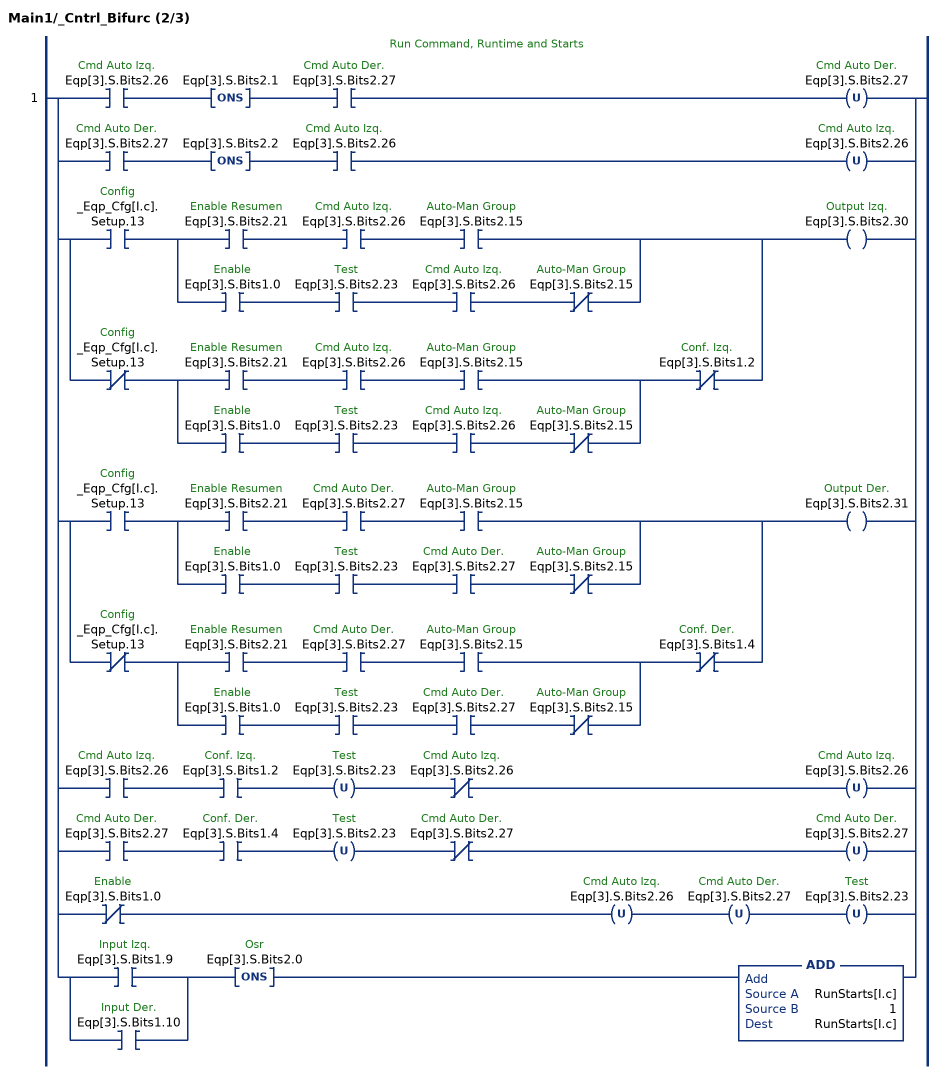
   // Run Command, Runtime and Starts
   1: [[XIC(Eqp[3].S.Bits2.26) ONS(Eqp[3].S.Bits2.1) XIC(Eqp[3].S.Bits2.27) OTU(Eqp[3].S.Bits2.27) ,XIC(Eqp[3].S.Bits2.27) ONS(Eqp[3].S.Bits2.2) XIC(Eqp[3].S.Bits2.26) OTU(Eqp[3].S.Bits2.26) ] ,[XIC(_Eqp_Cfg[I.c].Setup.13) [XIC(Eqp[3].S.Bits2.21) XIC(Eqp[3].S.Bits2.26) XIC(Eqp[3].S.Bits2.15) ,XIC(Eqp[3].S.Bits1.0) XIC(Eqp[3].S.Bits2.23) XIC(Eqp[3].S.Bits2.26) XIO(Eqp[3].S.Bits2.15) ] ,XIO(_Eqp_Cfg[I.c].Setup.13) [XIC(Eqp[3].S.Bits2.21) XIC(Eqp[3].S.Bits2.26) XIC(Eqp[3].S.Bits2.15) ,XIC(Eqp[3].S.Bits1.0) XIC(Eqp[3].S.Bits2.23) XIC(Eqp[3].S.Bits2.26) XIO(Eqp[3].S.Bits2.15) ] XIO(Eqp[3].S.Bits1.2) ] OTE(Eqp[3].S.Bits2.30) ,[XIC(_Eqp_Cfg[I.c].Setup.13) [XIC(Eqp[3].S.Bits2.21) XIC(Eqp[3].S.Bits2.27) XIC(Eqp[3].S.Bits2.15) ,XIC(Eqp[3].S.Bits1.0) XIC(Eqp[3].S.Bits2.23) XIC(Eqp[3].S.Bits2.27) XIO(Eqp[3].S.Bits2.15) ] ,XIO(_Eqp_Cfg[I.c].Setup.13) [XIC(Eqp[3].S.Bits2.21) XIC(Eqp[3].S.Bits2.27) XIC(Eqp[3].S.Bits2.15) ,XIC(Eqp[3].S.Bits1.0) XIC(Eqp[3].S.Bits2.23) XIC(Eqp[3].S.Bits2.27) XIO(Eqp[3].S.Bits2.15) ] XIO(Eqp[3].S.Bits1.4) ] OTE(Eqp[3].S.Bits2.31) ,[XIC(Eqp[3].S.Bits2.26) XIC(Eqp[3].S.Bits1.2) OTU(Eqp[3].S.Bits2.23) XIO(Eqp[3].S.Bits2.26) OTU(Eqp[3].S.Bits2.26) ,XIC(Eqp[3].S.Bits2.27) XIC(Eqp[3].S.Bits1.4) OTU(Eqp[3].S.Bits2.23) XIO(Eqp[3].S.Bits2.27) OTU(Eqp[3].S.Bits2.27) ] ,XIO(Eqp[3].S.Bits1.0) OTU(Eqp[3].S.Bits2.26) OTU(Eqp[3].S.Bits2.27) OTU(Eqp[3].S.Bits2.23) ,[XIC(Eqp[3].S.Bits1.9) ,XIC(Eqp[3].S.Bits1.10) ] ONS(Eqp[3].S.Bits2.0) ADD(RunStarts[I.c],1,RunStarts[I.c]) ];
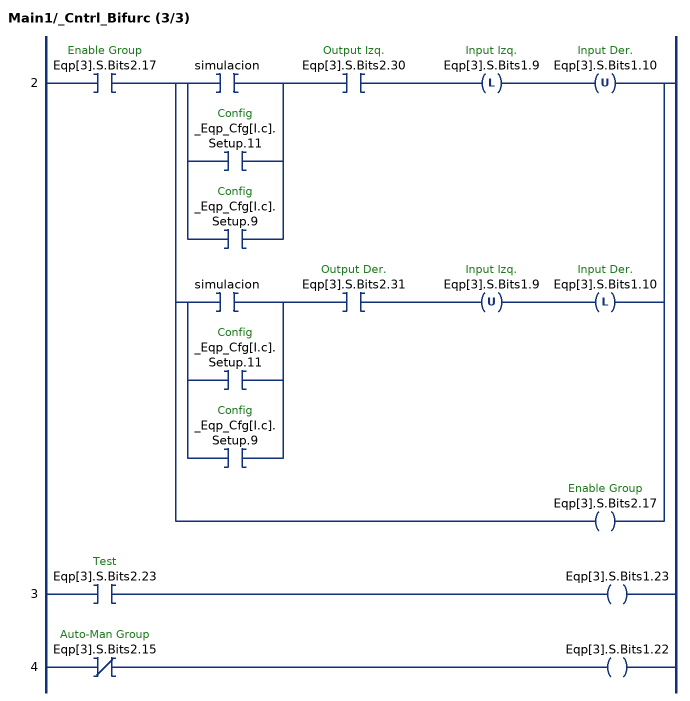
   2: XIC(Eqp[3].S.Bits2.17)[[XIC(simulacion) ,XIC(_Eqp_Cfg[I.c].Setup.11) ,XIC(_Eqp_Cfg[I.c].Setup.9) ] XIC(Eqp[3].S.Bits2.30) OTL(Eqp[3].S.Bits1.9) OTU(Eqp[3].S.Bits1.10) ,[XIC(simulacion) ,XIC(_Eqp_Cfg[I.c].Setup.11) ,XIC(_Eqp_Cfg[I.c].Setup.9) ] XIC(Eqp[3].S.Bits2.31) OTU(Eqp[3].S.Bits1.9) OTL(Eqp[3].S.Bits1.10) ,OTE(Eqp[3].S.Bits2.17) ];
   3: XIC(Eqp[3].S.Bits2.23)OTE(Eqp[3].S.Bits1.23);
   4: XIO(Eqp[3].S.Bits2.15)OTE(Eqp[3].S.Bits1.22);
END_ROUTINE
